// TIA Portal V20 export
DATA_BLOCK "ControlNodes"   // DB94
// stored: MemoryReserve 100, Namespace Unit1.Em9
   VAR
      em : "LAF_typeEmControlNode";
      emstate { S7_SetPoint := 'True'} : "LUC_typeStates";
      cm : "Unit1.Em9.typeCmControlNode";
      citiMap : Struct
         PMC : "LER_PMC_Input_Data";
         FlexNet { S7_SetPoint := 'True'} : "LER_FlexNet_Data";
      END_STRUCT;
      vision : "Unit1.Em9.typeSequenceControlNode";
      GRnR_vision { S7_SetPoint := 'True'} : "Unit1.Em9.typeSequenceControlNode_GRnR";
      emData : "LER_typePartData";
      SpecialFunctionMode : Struct
         DryRun : Struct
            JRdetectPV : Array[0..15] of Bool;
         END_STRUCT;
      END_STRUCT;
      cmVisionJRDetect : "LBC_typeDigitalSignalControlNode";
      cmVisionStageLiftUpDown : "LBC_typeTwoWayActuatorControlNode";
      cmVisionLightUpDown : "LBC_typeTwoWayActuatorControlNode";
      cmVisionControl : "LER_typeVisionControlNode";
   END_VAR
BEGIN
END_DATA_BLOCK
